FUNCTION_BLOCK ClockCounter
  (* Standard: 61499-2 *)
  (* Version 0.0, 2010-02-06, XPMUser, nxtControl GmbH, Template *)
  (* Compiler header: package fb.rt.cs725; *)
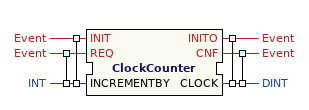
  EVENT_INPUT
    INIT WITH INCREMENTBY; (* Initialization Request *)
    REQ WITH INCREMENTBY; (* Normal Execution Request *)
  END_EVENT
  EVENT_OUTPUT
    INITO WITH CLOCK; (* Initialization Confirm *)
    CNF WITH CLOCK; (* Execution Confirmation *)
  END_EVENT
  VAR_INPUT
    INCREMENTBY : INT; (* Clock * ScaleUpFactor = CLOCK output *)
  END_VAR
  VAR_OUTPUT
    CLOCK : DINT; (* Output event qualifier *)
  END_VAR
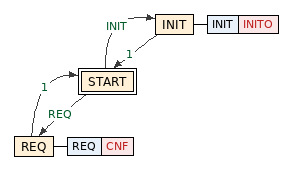
  EC_STATES
    START; (* Initial State *)
    INIT : INIT -> INITO; (* Initialization *)
    REQ : REQ -> CNF; (* Normal execution *)
  END_STATES
  EC_TRANSITIONS
    START TO INIT := INIT;
    INIT TO START := 1;
    START TO REQ := REQ;
    REQ TO START := 1;
  END_TRANSITIONS
  ALGORITHM INIT IN ST: (* Initialization algorithm *)
CLOCK := 0;
  END_ALGORITHM
  ALGORITHM REQ IN ST: (* Normally executed algorithm *)
CLOCK := CLOCK + (INCREMENTBY);

IF CLOCK >= 10000 THEN
  CLOCK := 1;
END_IF;
  END_ALGORITHM
END_FUNCTION_BLOCK
